PROGRAM MAIN
VAR
	
END_VAR

Making_Coffee(Grinding := GVL.GrindButton, ToastState := GVL.ToastState, GetOffBed := GVL.Wakeup, HeatButton := GVL.HeatingUp, Start := GVL.ix_Start, CoffeeMakingState => GVL.CoffeeState);
Making_Toast(LeverDown := GVL.LeverButton, BreadInserted := GVL.InsertedButton, CoffeeState := GVL.CoffeeState, MakingToastState => GVL.ToastState);

END_PROGRAM

(* stored: Version 1.1.0.1, ProductVersion 3.1.4024.15
   POU MAIN: Id {4f5b4da9-0ef4-4686-bbe2-392a45f36b5e}, SpecialFunc None *)
